// TIA Portal V19 export
DATA_BLOCK "DEV_7"   // DB5
{ S7_Optimized_Access := 'TRUE' }
// stored: MemoryReserve 0
   VAR
      Convoyer : "ModuleConvoyer";
   END_VAR
   VAR RETAIN
      Retains : Struct
         ConvoyerA : Struct
            ProducedUnits : DInt;
            "Type" : SInt;
         END_STRUCT;
         ConvoyerB : Struct
            ProducedUnits : DInt;
            "Type" : SInt;
         END_STRUCT;
      END_STRUCT;
      Recipes : Struct
         Convoyer : Struct
            "A" : Struct
               "Type" : SInt;
               StampingPL : Struct
                  Enable : Bool := TRUE;
                  Double : Bool;
                  SecondPush : Bool;
                  SecondPreasure : Real;
                  RegularPreasure : Real := 1.3;
                  MaxPreasure : Real := 4.0;
                  TimerMaxPreasure : Time := T#1300ms;
                  TimerStamping : Time := T#400ms;
                  TimerSecond : Time;
               END_STRUCT;
               SettingsPL : Struct
                  Camera : Bool := TRUE;
                  Blow : Bool := TRUE;
                  BlowTime : Time := T#1000ms;
               END_STRUCT;
               StampingCN : Struct
                  Enable : Bool := TRUE;
                  Double : Bool;
                  SecondPush : Bool := TRUE;
                  SecondPreasure : Real := 4.0;
                  RegularPreasure : Real := 1.3;
                  MaxPreasure : Real := 4.5;
                  TimerMaxPreasure : Time := T#1300ms;
                  TimerStamping : Time := T#800ms;
                  TimerSecond : Time := T#500ms;
               END_STRUCT;
               SettingsCN : Struct
                  Camera : Bool := TRUE;
                  Blow : Bool := TRUE;
                  BlowTime : Time := T#1000ms;
               END_STRUCT;
               StampingPlastic : Struct
                  Enable : Bool := TRUE;
                  Double : Bool;
                  SecondPush : Bool;
                  SecondPreasure : Real;
                  RegularPreasure : Real := 1.3;
                  MaxPreasure : Real := 4.0;
                  TimerMaxPreasure : Time := T#1300ms;
                  TimerStamping : Time := T#400ms;
                  TimerSecond : Time;
               END_STRUCT;
               SettingsPlastic : Struct
                  Camera : Bool := TRUE;
                  Blow : Bool := TRUE;
                  BlowTime : Time := T#1000ms;
               END_STRUCT;
               StampingTransport : Struct
                  Enable : Bool := FALSE;
                  Double : Bool := FALSE;
                  SecondPush : Bool := FALSE;
                  SecondPreasure : Real;
                  RegularPreasure : Real := 1.3;
                  MaxPreasure : Real := 4.0;
                  TimerMaxPreasure : Time := T#1300ms;
                  TimerStamping : Time := T#400ms;
                  TimerSecond : Time;
               END_STRUCT;
               SettingsTransport : Struct
                  Camera : Bool := FALSE;
                  Blow : Bool := FALSE;
                  BlowTime : Time := T#1000ms;
               END_STRUCT;
            END_STRUCT;
            "B" : Struct
               "Type" : SInt;
               StampingPL : Struct
                  Enable : Bool := TRUE;
                  Double : Bool;
                  SecondPush : Bool;
                  SecondPreasure : Real;
                  RegularPreasure : Real := 1.3;
                  MaxPreasure : Real := 4.0;
                  TimerMaxPreasure : Time := T#1300ms;
                  TimerStamping : Time := T#400ms;
                  TimerSecond : Time;
               END_STRUCT;
               SettingsPL : Struct
                  Camera : Bool := TRUE;
                  Blow : Bool := TRUE;
                  BlowTime : Time := T#1000ms;
               END_STRUCT;
               StampingCN : Struct
                  Enable : Bool := TRUE;
                  Double : Bool;
                  SecondPush : Bool := TRUE;
                  SecondPreasure : Real := 4.0;
                  RegularPreasure : Real := 1.3;
                  MaxPreasure : Real := 4.5;
                  TimerMaxPreasure : Time := T#1300ms;
                  TimerStamping : Time := T#800ms;
                  TimerSecond : Time := T#500ms;
               END_STRUCT;
               SettingsCN : Struct
                  Camera : Bool := TRUE;
                  Blow : Bool := TRUE;
                  BlowTime : Time := T#1000ms;
               END_STRUCT;
               StampingPlastic : Struct
                  Enable : Bool := TRUE;
                  Double : Bool;
                  SecondPush : Bool;
                  SecondPreasure : Real;
                  RegularPreasure : Real := 1.3;
                  MaxPreasure : Real := 4.0;
                  TimerMaxPreasure : Time := T#1300ms;
                  TimerStamping : Time := T#400ms;
                  TimerSecond : Time;
               END_STRUCT;
               SettingsPlastic : Struct
                  Camera : Bool := TRUE;
                  Blow : Bool := TRUE;
                  BlowTime : Time := T#1000ms;
               END_STRUCT;
               StampingTransport : Struct
                  Enable : Bool := FALSE;
                  Double : Bool := FALSE;
                  SecondPush : Bool := FALSE;
                  SecondPreasure : Real;
                  RegularPreasure : Real := 1.3;
                  MaxPreasure : Real := 4.0;
                  TimerMaxPreasure : Time := T#1300ms;
                  TimerStamping : Time := T#400ms;
                  TimerSecond : Time;
               END_STRUCT;
               SettingsTransport : Struct
                  Camera : Bool := FALSE;
                  Blow : Bool := FALSE;
                  BlowTime : Time := T#1000ms;
               END_STRUCT;
            END_STRUCT;
         END_STRUCT;
      END_STRUCT;
      OPC : Struct
         Convoyer : Struct
            "A" : Struct
               LifetimeProduction : DInt;
               CycleTime : Time;
               CameraCycle : Time;
               StampingCycle : Time;
               ActualRecipe : WString[30];
               Status : Struct
                  ReadyToWork : Bool;
                  Working : Bool;
                  Error : Bool;
               END_STRUCT;
            END_STRUCT;
            "B" : Struct
               LifetimeProduction : DInt;
               CycleTime : Time;
               CameraCycle : Time;
               StampingCycle : Time;
               ActualRecipe : WString[30];
               Status : Struct
                  ReadyToWork : Bool;
                  Working : Bool;
                  Error : Bool;
               END_STRUCT;
            END_STRUCT;
         END_STRUCT;
      END_STRUCT;
   END_VAR
BEGIN
   Convoyer.Modular_A.CameraConnection.InterfaceId := 64;
   Convoyer.Modular_A.CameraConnection.ID := 1;
   Convoyer.Modular_A.CameraConnection.ConnectionType := 16#0B;
   Convoyer.Modular_A.CameraConnection.ActiveEstablished := false;
   Convoyer.Modular_A.CameraConnection.RemoteAddress.ADDR[1] := 192;
   Convoyer.Modular_A.CameraConnection.RemoteAddress.ADDR[2] := 168;
   Convoyer.Modular_A.CameraConnection.RemoteAddress.ADDR[3] := 0;
   Convoyer.Modular_A.CameraConnection.RemoteAddress.ADDR[4] := 70;
   Convoyer.Modular_A.CameraConnection.RemotePort := 0;
   Convoyer.Modular_A.CameraConnection.LocalPort := 2137;
   Convoyer.Modular_A.Pneumatics.Stamping.Timers.In := T#6000ms;
   Convoyer.Modular_A.Pneumatics.Stamping.Timers.Out := T#5000ms;
   Convoyer.Modular_A.Pneumatics.IVT.Sensor.Analog.SetValue := 0.0;
   Convoyer.Modular_A.Pneumatics.IVT.Sensor.Settings.Min := 0.0;
   Convoyer.Modular_A.Pneumatics.IVT.Sensor.Settings.Max := 7.0;
   Convoyer.Modular_A.HMI.Camera.Enable := TRUE;
   Convoyer.Modular_A.HMI.Camera.TimerConnection := T#100000ms;
   Convoyer.Modular_A.HMI.Stamping.Enable := TRUE;
   Convoyer.Modular_A.HMI.Stamping.RegularPreasure := 3.0;
   Convoyer.Modular_A.HMI.Stamping.MaxPreasure := 6.0;
   Convoyer.Modular_A.HMI.Stamping.TimerMaxPreasure := T#1500ms;
   Convoyer.Modular_A.HMI.Stamping.TimerStamping := T#1000ms;
   Convoyer.Modular_A.HMI.Blow.Enable := TRUE;
   Convoyer.Modular_A.HMI.Blow."Time" := T#1000ms;
   Convoyer.Modular_B.CameraConnection.InterfaceId := 64;
   Convoyer.Modular_B.CameraConnection.ID := 16#2;
   Convoyer.Modular_B.CameraConnection.ConnectionType := 16#0B;
   Convoyer.Modular_B.CameraConnection.ActiveEstablished := FALSE;
   Convoyer.Modular_B.CameraConnection.RemoteAddress.ADDR[1] := 192;
   Convoyer.Modular_B.CameraConnection.RemoteAddress.ADDR[2] := 168;
   Convoyer.Modular_B.CameraConnection.RemoteAddress.ADDR[3] := 0;
   Convoyer.Modular_B.CameraConnection.RemoteAddress.ADDR[4] := 71;
   Convoyer.Modular_B.CameraConnection.RemotePort := 0;
   Convoyer.Modular_B.CameraConnection.LocalPort := 2137;
END_DATA_BLOCK
